PROGRAM MAIN
VAR
END_VAR

RunGrindingWheel();

END_PROGRAM

(* stored: Version 1.1.0.1, ProductVersion 3.1.4024.12
   POU MAIN: Id {6e837af7-6a90-49c7-bd59-7eab18a01e98}, SpecialFunc None *)
